# EPICS substitutions: HVCAENx527App/Db/HVCAENx527ch.substitutions
file "$(TOP)/templates/HVCAENx527ch.tpl" {
	pattern {PSNAME,CHANNUM,CHADDR}
	{"\$(P):\$(PSNAME):\$(SLOT)","\$(CHANNUM)","\$(CHADDR)"}
}
